// Mitsubishi GX Developer project: 16-403   PLC: FX3G

PROGRAM MAIN
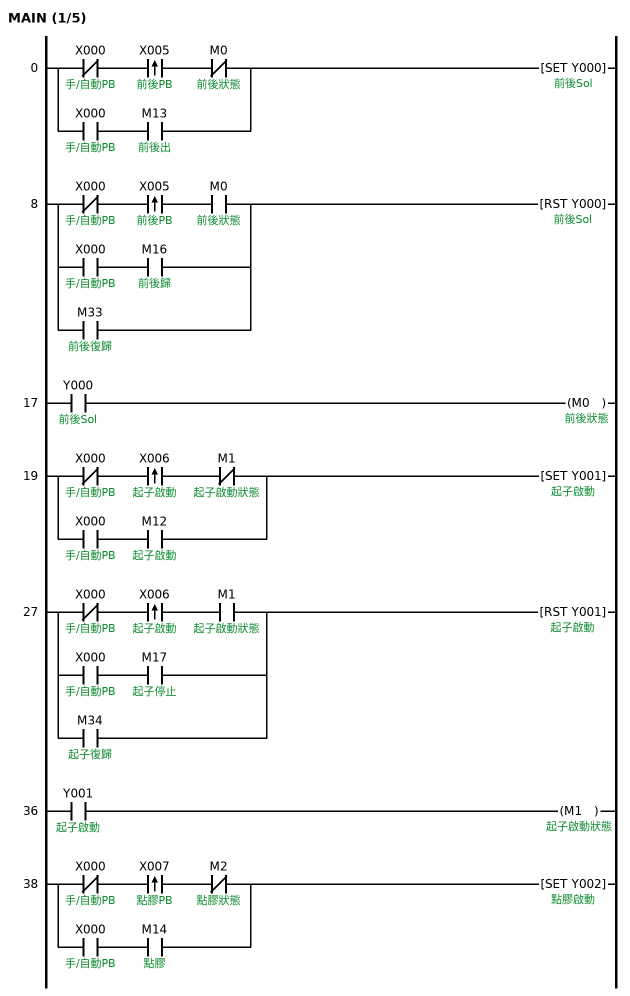
0     LDI     X000  ; 手/自動PB
      ANDP    X005  ; 前後PB
      ANI     M0  ; 前後狀態
      LD      X000  ; 手/自動PB
      AND     M13  ; 前後出
      ORB
      SET     Y000  ; 前後Sol
8     LDI     X000  ; 手/自動PB
      ANDP    X005  ; 前後PB
      AND     M0  ; 前後狀態
      LD      X000  ; 手/自動PB
      AND     M16  ; 前後歸
      ORB
      OR      M33  ; 前後復歸
      RST     Y000  ; 前後Sol
17    LD      Y000  ; 前後Sol
      OUT     M0  ; 前後狀態
19    LDI     X000  ; 手/自動PB
      ANDP    X006  ; 起子啟動
      ANI     M1  ; 起子啟動狀態
      LD      X000  ; 手/自動PB
      AND     M12  ; 起子啟動
      ORB
      SET     Y001  ; 起子啟動
27    LDI     X000  ; 手/自動PB
      ANDP    X006  ; 起子啟動
      AND     M1  ; 起子啟動狀態
      LD      X000  ; 手/自動PB
      AND     M17  ; 起子停止
      ORB
      OR      M34  ; 起子復歸
      RST     Y001  ; 起子啟動
36    LD      Y001  ; 起子啟動
      OUT     M1  ; 起子啟動狀態
38    LDI     X000  ; 手/自動PB
      ANDP    X007  ; 點膠PB
      ANI     M2  ; 點膠狀態
      LD      X000  ; 手/自動PB
      AND     M14  ; 點膠
      ORB
      SET     Y002  ; 點膠啟動
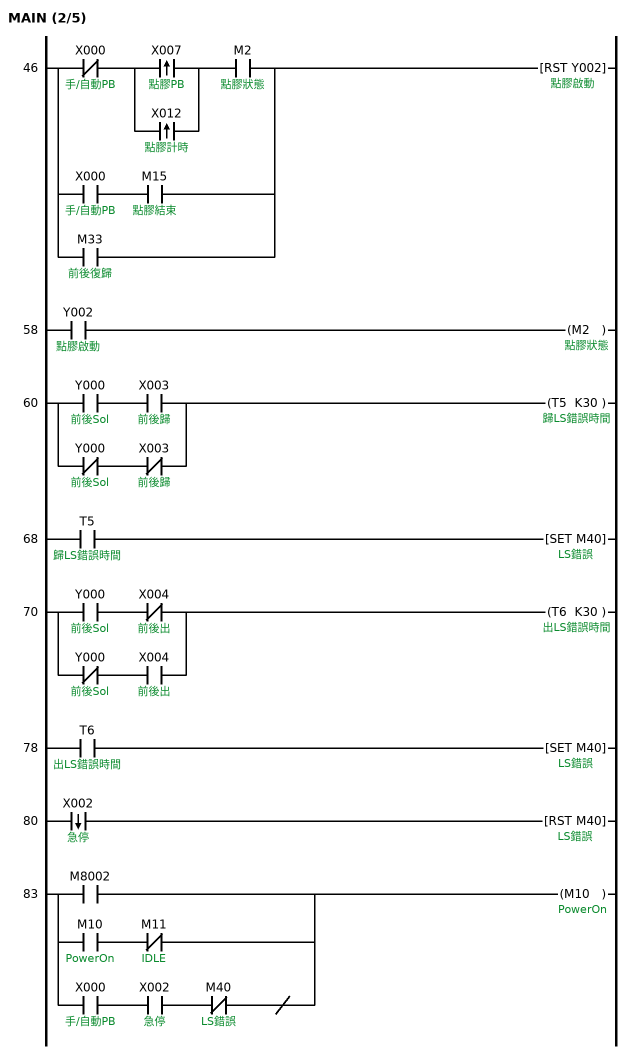
46    LDI     X000  ; 手/自動PB
      LDP     X007  ; 點膠PB
      ORP     X012  ; 點膠計時
      ANB
      AND     M2  ; 點膠狀態
      LD      X000  ; 手/自動PB
      AND     M15  ; 點膠結束
      ORB
      OR      M33  ; 前後復歸
      RST     Y002  ; 點膠啟動
58    LD      Y002  ; 點膠啟動
      OUT     M2  ; 點膠狀態
60    LD      Y000  ; 前後Sol
      AND     X003  ; 前後歸
      LDI     Y000  ; 前後Sol
      ANI     X003  ; 前後歸
      ORB
      OUT     T5 K30  ; 歸LS錯誤時間
68    LD      T5  ; 歸LS錯誤時間
      SET     M40  ; LS錯誤
70    LD      Y000  ; 前後Sol
      ANI     X004  ; 前後出
      LDI     Y000  ; 前後Sol
      AND     X004  ; 前後出
      ORB
      OUT     T6 K30  ; 出LS錯誤時間
78    LD      T6  ; 出LS錯誤時間
      SET     M40  ; LS錯誤
80    LDF     X002  ; 急停
      RST     M40  ; LS錯誤
83    LD      M8002
      LD      M10  ; PowerOn
      ANI     M11  ; IDLE
      ORB
      LD      X000  ; 手/自動PB
      AND     X002  ; 急停
      ANI     M40  ; LS錯誤
      INV
      ORB
      OUT     M10  ; PowerOn
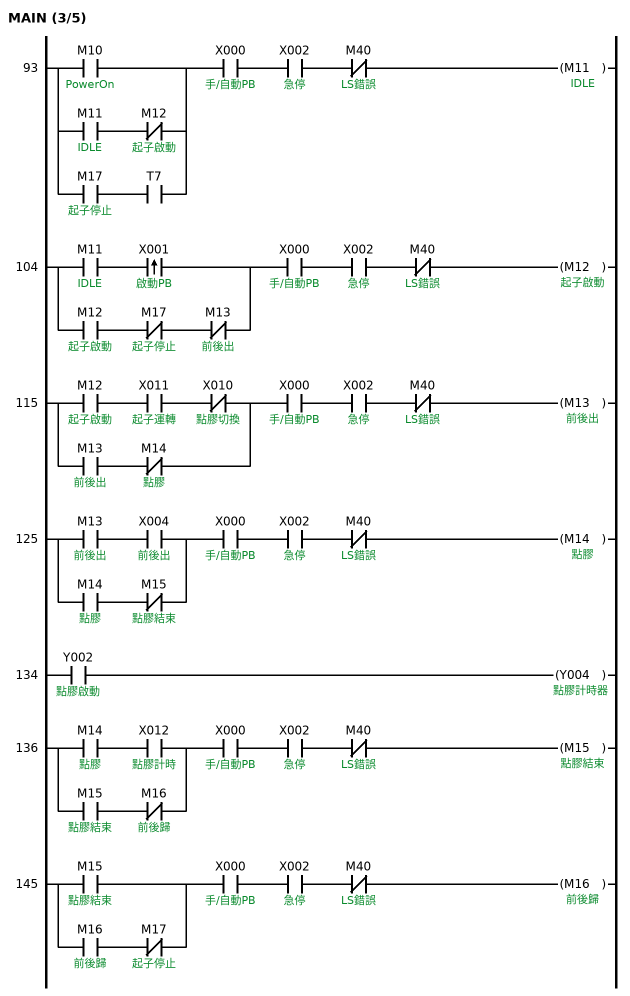
93    LD      M10  ; PowerOn
      LD      M11  ; IDLE
      ANI     M12  ; 起子啟動
      ORB
      LD      M17  ; 起子停止
      AND     T7
      ORB
      AND     X000  ; 手/自動PB
      AND     X002  ; 急停
      ANI     M40  ; LS錯誤
      OUT     M11  ; IDLE
104   LD      M11  ; IDLE
      ANDP    X001  ; 啟動PB
      LD      M12  ; 起子啟動
      ANI     M17  ; 起子停止
      ANI     M13  ; 前後出
      ORB
      AND     X000  ; 手/自動PB
      AND     X002  ; 急停
      ANI     M40  ; LS錯誤
      OUT     M12  ; 起子啟動
115   LD      M12  ; 起子啟動
      AND     X011  ; 起子運轉
      ANI     X010  ; 點膠切換
      LD      M13  ; 前後出
      ANI     M14  ; 點膠
      ORB
      AND     X000  ; 手/自動PB
      AND     X002  ; 急停
      ANI     M40  ; LS錯誤
      OUT     M13  ; 前後出
125   LD      M13  ; 前後出
      AND     X004  ; 前後出
      LD      M14  ; 點膠
      ANI     M15  ; 點膠結束
      ORB
      AND     X000  ; 手/自動PB
      AND     X002  ; 急停
      ANI     M40  ; LS錯誤
      OUT     M14  ; 點膠
134   LD      Y002  ; 點膠啟動
      OUT     Y004  ; 點膠計時器
136   LD      M14  ; 點膠
      AND     X012  ; 點膠計時
      LD      M15  ; 點膠結束
      ANI     M16  ; 前後歸
      ORB
      AND     X000  ; 手/自動PB
      AND     X002  ; 急停
      ANI     M40  ; LS錯誤
      OUT     M15  ; 點膠結束
145   LD      M15  ; 點膠結束
      LD      M16  ; 前後歸
      ANI     M17  ; 起子停止
      ORB
      AND     X000  ; 手/自動PB
      AND     X002  ; 急停
      ANI     M40  ; LS錯誤
      OUT     M16  ; 前後歸
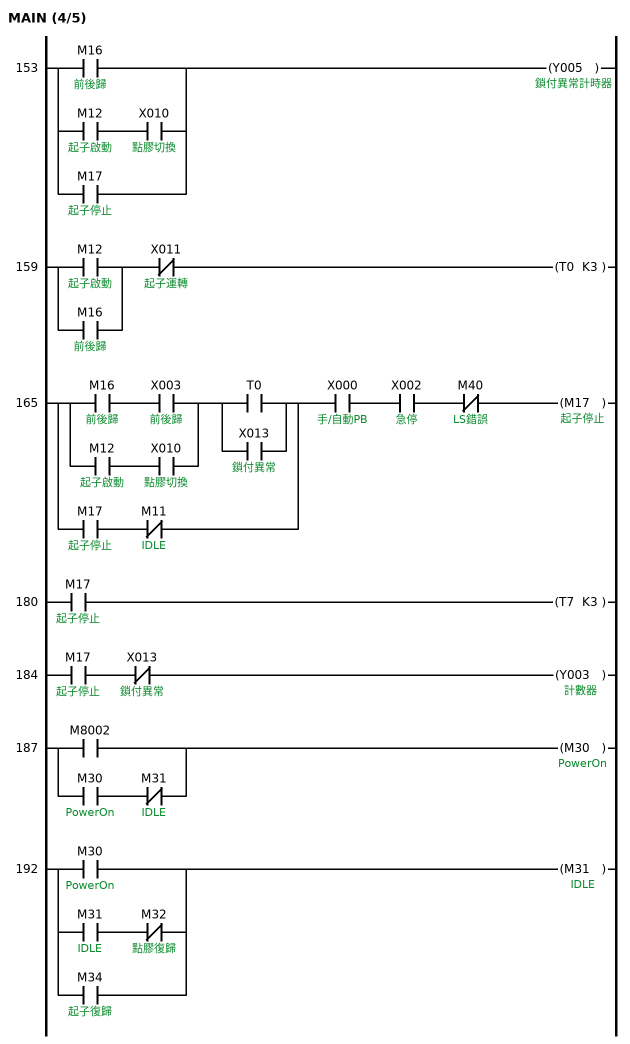
153   LD      M16  ; 前後歸
      LD      M12  ; 起子啟動
      AND     X010  ; 點膠切換
      ORB
      OR      M17  ; 起子停止
      OUT     Y005  ; 鎖付異常計時器
159   LD      M12  ; 起子啟動
      OR      M16  ; 前後歸
      ANI     X011  ; 起子運轉
      OUT     T0 K3
165   LD      M16  ; 前後歸
      AND     X003  ; 前後歸
      LD      M12  ; 起子啟動
      AND     X010  ; 點膠切換
      ORB
      LD      T0
      OR      X013  ; 鎖付異常
      ANB
      LD      M17  ; 起子停止
      ANI     M11  ; IDLE
      ORB
      AND     X000  ; 手/自動PB
      AND     X002  ; 急停
      ANI     M40  ; LS錯誤
      OUT     M17  ; 起子停止
180   LD      M17  ; 起子停止
      OUT     T7 K3
184   LD      M17  ; 起子停止
      ANI     X013  ; 鎖付異常
      OUT     Y003  ; 計數器
187   LD      M8002
      LD      M30  ; PowerOn
      ANI     M31  ; IDLE
      ORB
      OUT     M30  ; PowerOn
192   LD      M30  ; PowerOn
      LD      M31  ; IDLE
      ANI     M32  ; 點膠復歸
      ORB
      OR      M34  ; 起子復歸
      OUT     M31  ; IDLE
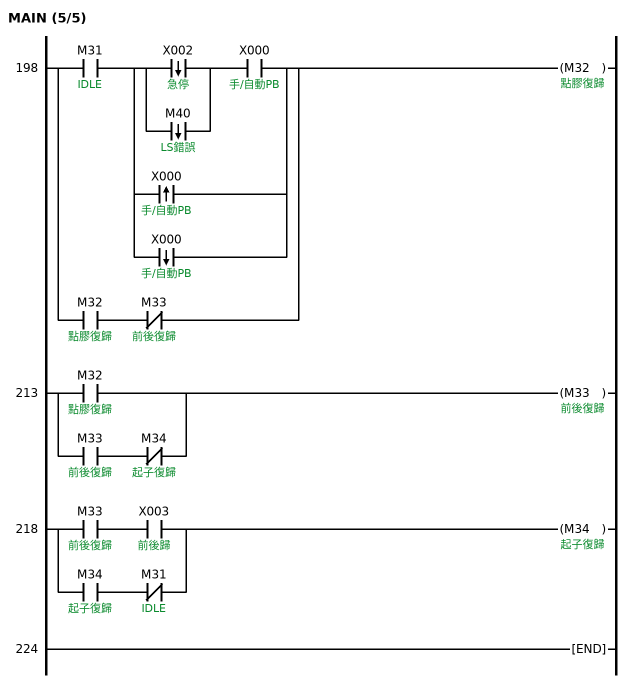
198   LD      M31  ; IDLE
      LDF     X002  ; 急停
      ORF     M40  ; LS錯誤
      AND     X000  ; 手/自動PB
      ORP     X000  ; 手/自動PB
      ORF     X000  ; 手/自動PB
      ANB
      LD      M32  ; 點膠復歸
      ANI     M33  ; 前後復歸
      ORB
      OUT     M32  ; 點膠復歸
213   LD      M32  ; 點膠復歸
      LD      M33  ; 前後復歸
      ANI     M34  ; 起子復歸
      ORB
      OUT     M33  ; 前後復歸
218   LD      M33  ; 前後復歸
      AND     X003  ; 前後歸
      LD      M34  ; 起子復歸
      ANI     M31  ; IDLE
      ORB
      OUT     M34  ; 起子復歸
224   END
END_PROGRAM

// device comments not shown above
M20  ; 不點膠
Y006  ; 起子電源
T1  ; 起子啟動時間
T2  ; 完成時間
